{attribute 'qualified_only'}
{attribute 'strict'}
TYPE AirPressureStatus :
(
	UNKNOWN := 0,
	ERROR	:= 1,
	WARNING := 2,          
    HEALTH  := 3,      
    OVERTOP := 4       

);
END_TYPE

(* stored: Version 1.1.0.1, ProductVersion 3.1.4024.12
   DUT AirPressureStatus: Id {b4f6917d-b4e8-410e-a1c1-448b6eb74fcc} *)
